// TIA Portal V19 export
DATA_BLOCK "A02_DEBUG"   // DB196
// stored: MemoryReserve 100
   VAR
      Force_Sinamics_CtrlSafe : Bool := FALSE;
      Forse_Contactors_CtrlSafe : Bool := FALSE;
      MatPresence_Entry : Bool := FALSE;
      MatPresence_BeforeMW : Bool := FALSE;
      MatPresence_AfterMW : Bool := FALSE;
      MatPresence_AfterFAK : Bool := FALSE;
      CutEnableDebug : Bool := FALSE;
      CutToDO : Int := 0;
   END_VAR
   VAR RETAIN
      CutDone : Int := 174;
      MetersDone : LReal := 472013.010252576;
   END_VAR
   VAR
      MoveTrk : Bool := FALSE;
      WeldDone : Bool := FALSE;
      SetWrongCut : Bool := FALSE;
      MwFakCalc : Struct
         GripperPosRel : LReal := 0.0;
      END_STRUCT;
      MAchineAborting : Struct
         RollformingMng : Bool := FALSE;
         FakCalc : Bool := FALSE;
         Weldreg : Bool := FALSE;
         A02_HU : Bool := FALSE;
         RegolazioneFormato : Bool := FALSE;
         PitTable : Bool := FALSE;
         Rollformer : Bool := FALSE;
         RollformerLubr : Bool := FALSE;
         FlyingCarriage : Bool := FALSE;
         CarriageLubr : Bool := FALSE;
         FinalCut : Bool := FALSE;
         FinalCutLubr : Bool := FALSE;
         Accroll : Bool := FALSE;
         AreaGen : Bool := FALSE;
         Loop1 : Bool := FALSE;
      END_STRUCT;
      MachineAlarm : Int := 0;
      PosAxToPosMat : Struct
         PosAx : LReal := 0.0;
         PosMatCalculated : LReal := 169629.13183459;
      END_STRUCT;
      PosMatToPosAx : Struct
         PosMat : LReal := 0.0;
         PosAxCalculated : LReal := 830413.680811859;
      END_STRUCT;
      StopDaMes : Struct
         STOP_Part_Recondition : Bool := FALSE;
         STOP_Order_Complete : Bool := FALSE;
         STOP_O_ACT_Empty : Bool := FALSE;
         STOP_End_Of_Proroduction : Bool := FALSE;
         STOP_FineTurno : Bool := FALSE;
         STOP_ControlloQualita : Bool := FALSE;
         Stop_Matrice_Colata_Coil : Bool := FALSE;
      END_STRUCT;
   END_VAR
BEGIN
END_DATA_BLOCK
